Fanuc KAREL source: IO0186.KL

-- PROVISIONAL review KL for V770-1; original PC SHA256 2182ecd7e29cc3fec465617e329c668065931b6ea44d808c65776ee3dc8761b7
-- Incomplete behavior may be omitted. Consult companion uncertainty JSON. Do not deploy.
PROGRAM IO0186
%NOLOCKGROUP
-- UNRESOLVED_LOCAL_POOL 5 cells at code offset 13; source declarations unknown
-- DIRECT_LOCAL_WORD_ACCESS alone does not prove INTEGER, REAL, or BOOLEAN
BEGIN
  -- UNRESOLVED_PC offsets 0-18; opcodes 2B,2C,7B
  -- UNRESOLVED_PC offsets 23-30; opcodes 9D,23
  -- UNRESOLVED_PC offsets 35-49; opcodes 2E,22,9D,33,35
  -- UNRESOLVED_PC offsets 54-61; opcodes 9D,23
  -- UNRESOLVED_PC offsets 66-77; opcodes 2E,23
  -- UNRESOLVED_PC offsets 82-102; opcodes 9D,19,9D,57,2E,19,9C,57,46,79
  -- UNRESOLVED_PC offsets 107-121; opcodes 21,9D,52,23
  -- UNRESOLVED_PC offsets 131-135; opcodes 7F
  -- UNRESOLVED_PC offsets 140-144; opcodes 27,AA
  -- UNRESOLVED_PC offsets 149-153; opcodes 7F
END IO0186
